(*!
<summary>Exposes a task-driven timer's interval, observations and restart operation.</summary>
<description>
Drive the timer through the inherited task lifecycle. Reading observations does not advance time; the
implementation updates them while executing. Timer-specific TON behavior is documented by Timer.
</description>
*)
INTERFACE ITimer EXTENDS TOF_Tasks.ITask

{attribute 'monitoring' := 'call'}
(*!
<summary>Reports the timer's latest elapsed observation.</summary>
<description>
Reading does not update or consume the observation. For Timer this is TON.Q, retained after normal completion
until Reset or restart; it is not independently a successful task-completion result.
</description>
*)
PROPERTY Elapsed : BOOL
GET
END_GET
END_PROPERTY

{attribute 'monitoring' := 'call'}
(*!
<summary>Returns the latest elapsed-time observation without advancing the timer.</summary>
<description>
For Timer this is TON.ET from the most recent TON evaluation, not a live clock read. Reset clears the
observation.
</description>
*)
PROPERTY ElapsedTime : TIME
GET
END_GET
END_PROPERTY

{attribute 'monitoring' := 'call'}
(*!
<summary>Gets or sets the configured timer interval.</summary>
<description>
For Timer, assignment changes TON.PT without a reset, start or immediate observation update. Use
SetIntervalAndRestart to apply an interval and begin timing it from zero.
</description>
*)
PROPERTY Interval : TIME
GET
END_GET
SET
END_SET
END_PROPERTY

(*!
<summary>Prepare a restart, then set the interval and start timing immediately.</summary>
<description>
The method assigns the new interval only after stopping and Reset succeed. A refused preparation returns
FALSE without that assignment; partial effects of descendant callbacks are not rolled back. If Start fails
after preparation, the new interval remains configured. No deferred restart is scheduled. Call outside task
callbacks.
</description>
<param name="interval">Preset for the new run, including zero for completion on its first Execute.</param>
*)

METHOD SetIntervalAndRestart : BOOL
VAR_INPUT
	interval : TIME;
END_VAR
END_METHOD

(*!
<summary>Reports completion in the Execute that observes the timer elapsed.</summary>
<description>
For the ordinary Timer, includes a zero interval and adds no stopping cycle. Read after Execute. The pulse is
cleared by the next Execute, Reset or successful restart; reading does not consume it.
</description>
*)

{attribute 'monitoring' := 'call'}

PROPERTY Triggered : BOOL
GET
END_GET
END_PROPERTY

END_INTERFACE

(* stored: Version 1.1.0.1
   Itf ITimer: Id {48689db6-2a88-4baa-afb2-9879b912e6f4}
   Property Elapsed: Id {65834b8f-b730-4fea-9c2a-df9357a8a87e}
   Get Get: Id {5d233c01-dc6d-4140-812f-10b6675984d3}
   Property ElapsedTime: Id {6be46376-d7c5-403e-aee6-fae9d20ed935}
   Get Get: Id {86906748-573a-4363-89bf-e929ab4689a6}
   Property Interval: Id {9f58246e-11d4-40f2-bdfb-fcd044bf8727}
   Get Get: Id {9ce0c5a5-d97f-4b20-83a7-395189cc87b8}
   Set Set: Id {fde3a764-d52d-491a-83df-f731b46a066a}
   Method SetIntervalAndRestart: Id {c817cee2-d504-4502-8d64-33ad72dda540}
   Property Triggered: Id {62331caa-0a29-423d-9d27-d148f730ec3a}
   Get Get: Id {8093b050-d68f-420c-9a07-84bf79b0e4d3} *)
